Universal Robots PolyScope program: zaboj_fiala_program.urp

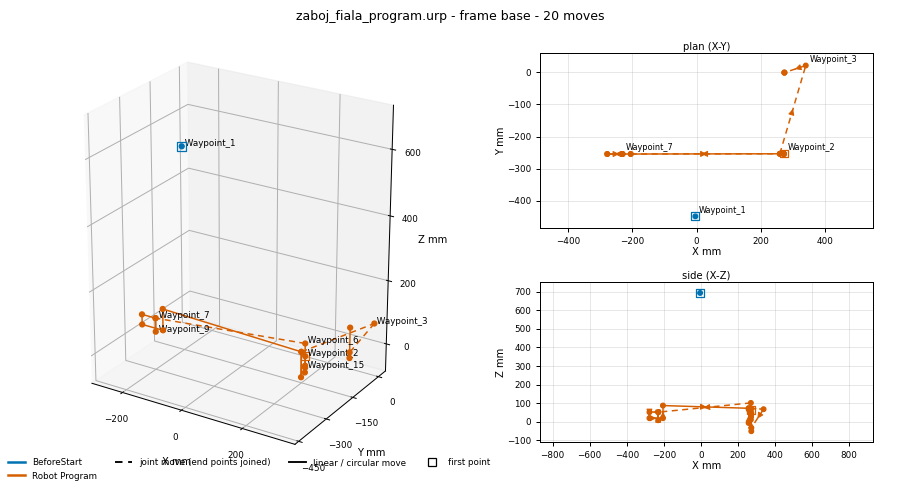
[picture p0: tool path of zaboj_fiala_program.urp in frame base, 20 of 20 moves have a stored position in this frame; points joined in program order, loops and branches not executed]
Program zaboj_fiala_program (installation=zaboj_fiala_instalace directory=/programs/usbdisk_0/new folder createdIn=5.21.2 lastSavedIn=5.21.2 robotSerialNumber=20185300578)
Calibrated DH parameters: a=[-0.000189, -0.243548, -0.212949, 0.000139, -0.000171, 0]; d=[0.151928, 2.340352, -3.79233, 1.582506, 0.085299, 0.092103]; alpha=[1.570802, 0.003282, -0.008312, 1.570809, -1.571939, 0]; deltaTheta=[0, 0.031526, 6.30827, -0.05661, 0, 0]
InitVariablesNode variables(variable(name=Pallet_1_cnt, expression=1), variable(name=Pallet_1_lct, expression=1), variable(name=Pallet_1_lno, expression=1), variable(name=Pallet_1_sep, expression=False), variable(name=Pallet_1_tct, expression=1), variable(name=qNearApproach, expression=[0,0,0,0,0,0]))
BeforeStart
  URCap Gripper Activate (Robotiq_Grippers, Robotiq Inc.) dataModel(ResetAndActivateKey=true)
  MoveJ speed 60 deg/s, acceleration 80 deg/s^2 (useActiveTCP=true optimoveEnabled=false optiMoveSpeed=0.3 optiMoveAcceleration=0.09) feature=Base
    Waypoint Waypoint_1: TCP in base x=-3.732 y=-447.764 z=694.669 mm, rx=0.0104 ry=2.2175 rz=-2.2154 rad; joints [0.253, -89.95, 0.625, -89.448, -0.524, -0.516] deg; TCP offset x=0.341 y=-0.738 z=225.168 mm, rx=0 ry=0 rz=-0.0028 rad
  Wait DigitalInput pin=digital_in[2]; digitalValue=1
Robot Program (runOnlyOnce=false)
  MoveJ speed 60 deg/s, acceleration 80 deg/s^2 (useActiveTCP=true optimoveEnabled=false optiMoveSpeed=0.3 optiMoveAcceleration=0.09) feature=Base
    Waypoint Waypoint_2: TCP in base x=270.562 y=-252.46 z=60.751 mm, rx=-2.2056 ry=2.2371 rz=0 rad; joints [-22.23, -101.243, -82.016, -86.674, 89.555, -21.444] deg
  Wait DigitalInput pin=digital_in[2]; digitalValue=1
  URCap Gripper (Robotiq_Grippers, Robotiq Inc.) dataModel(position=100.0, force=20.0, speed=100.0, positionInDouble=100.0, forceInDouble=20.0, speedInDouble=100.0, slaveIds=[9], blocking=true, robotCompliant=false)
  MoveL speed 50 mm/s, acceleration 1200 mm/s^2 (useActiveTCP=true optimoveEnabled=false optiMoveSpeed=0.01 optiMoveAcceleration=0.0001) feature=Base
    Waypoint Waypoint_15: TCP in base x=270.562 y=-252.46 z=25.108 mm, rx=-2.2056 ry=2.2371 rz=0 rad; joints [-22.21, -102.437, -90.223, -77.272, 89.565, -21.501] deg; TCP offset x=0.341 y=-0.738 z=225.168 mm, rx=0 ry=0 rz=-0.0028 rad
    var_1 := force()
    MoveL speed 250 mm/s, acceleration 1200 mm/s^2 (useActiveTCP=true optimoveEnabled=false optiMoveSpeed=0.3 optiMoveAcceleration=0.09) feature=Base
      Waypoint Waypoint_4: TCP in base x=271.723 y=-254.714 z=32.577 mm, rx=-2.2024 ry=2.234 rz=-0.0171 rad; joints [-22.478, -101.846, -89.192, -78.218, 89.558, -21.757] deg; TCP offset x=0.341 y=-0.738 z=225.168 mm, rx=0 ry=0 rz=-0.0028 rad
    If var_1>5
      MoveL speed 250 mm/s, acceleration 1200 mm/s^2 (useActiveTCP=true optimoveEnabled=false optiMoveSpeed=0.3 optiMoveAcceleration=0.09) feature=Base
        URCap Gripper (Robotiq_Grippers, Robotiq Inc.) dataModel(position=0.0, force=20.0, speed=100.0, positionInDouble=0.0, forceInDouble=20.0, speedInDouble=100.0, slaveIds=[9], blocking=true, robotCompliant=false)
        Waypoint Waypoint_5: TCP in base x=270.562 y=-253.262 z=10.468 mm, rx=-2.2056 ry=2.2371 rz=0 rad; joints [-22.326, -103.45, -93.013, -73.469, 89.574, -21.647] deg; TCP offset x=0.341 y=-0.738 z=225.168 mm, rx=0 ry=0 rz=-0.0028 rad
        URCap Gripper (Robotiq_Grippers, Robotiq Inc.) dataModel(position=100.0, force=20.0, speed=100.0, positionInDouble=100.0, forceInDouble=20.0, speedInDouble=100.0, slaveIds=[9], blocking=true, robotCompliant=false)
        SetPayload (workpieceName=Payload_brick payloadTransitionTime=0.05)
        Waypoint Waypoint_6: TCP in base x=270.562 y=-253.262 z=100.61 mm, rx=-2.2056 ry=2.2371 rz=0 rad; joints [-22.379, -101.712, -70.714, -97.506, 89.565, -21.504] deg
      MoveJ speed 60 deg/s, acceleration 80 deg/s^2 (useActiveTCP=true optimoveEnabled=false optiMoveSpeed=0.3 optiMoveAcceleration=0.09) feature=Base
        Waypoint Waypoint_7: TCP in base x=-230.059 y=-254.189 z=50.546 mm, rx=-2.2056 ry=2.2371 rz=0 rad; joints [-109.77, -94.859, -92.164, -82.912, 89.537, -109.018] deg
      MoveL speed 250 mm/s, acceleration 1200 mm/s^2 (useActiveTCP=true optimoveEnabled=false optiMoveSpeed=0.3 optiMoveAcceleration=0.09) feature=Base
        Waypoint Waypoint_9: TCP in base x=-230.059 y=-254.189 z=7.047 mm, rx=-2.2056 ry=2.2371 rz=0 rad; joints [-109.748, -97.199, -101.559, -71.177, 89.561, -109.091] deg
        URCap Gripper (Robotiq_Grippers, Robotiq Inc.) dataModel(position=0.0, force=100.0, speed=20.0, positionInDouble=0.0, forceInDouble=100.0, speedInDouble=20.0, slaveIds=[9], blocking=true, robotCompliant=false)
        SetPayload (workpieceName=Payload_Empty payloadTransitionTime=0.05)
        Waypoint Waypoint_7: TCP in base x=-230.059 y=-254.189 z=50.546 mm, rx=-2.2056 ry=2.2371 rz=0 rad; joints [-109.77, -94.859, -92.164, -82.912, 89.537, -109.018] deg
        URCap Gripper (Robotiq_Grippers, Robotiq Inc.) dataModel(position=100.0, force=100.0, speed=100.0, positionInDouble=100.0, forceInDouble=100.0, speedInDouble=100.0, slaveIds=[9], blocking=true, robotCompliant=false)
        MoveL speed 250 mm/s, acceleration 1200 mm/s^2 (useActiveTCP=true optimoveEnabled=false optiMoveSpeed=0.3 optiMoveAcceleration=0.09) feature=Base
          Waypoint Waypoint_11: motionParameters(blendRadius=0.01); TCP in base x=-277.401 y=-254.189 z=50.546 mm, rx=-2.2056 ry=2.2371 rz=0 rad; joints [-117.208, -103.279, -82.236, -84.42, 89.564, -116.439] deg
          Waypoint Waypoint_12: motionParameters(blendRadius=0.01); TCP in base x=-277.401 y=-254.189 z=18.071 mm, rx=-2.2056 ry=2.2371 rz=0 rad; joints [-117.19, -104.607, -89.405, -75.923, 89.576, -116.491] deg
          Waypoint Waypoint_13: motionParameters(blendRadius=0.01); TCP in base x=-204.474 y=-254.189 z=18.071 mm, rx=-2.2056 ry=2.2371 rz=0 rad; joints [-105.212, -92.223, -103.906, -73.805, 89.539, -104.534] deg
          Waypoint Waypoint_14: TCP in base x=-204.474 y=-254.189 z=86.413 mm, rx=-2.2056 ry=2.2371 rz=0 rad; joints [-105.25, -90.231, -87.365, -92.339, 89.523, -104.42] deg
    Else 
      MoveL speed 250 mm/s, acceleration 1200 mm/s^2 (useActiveTCP=true optimoveEnabled=false optiMoveSpeed=0.3 optiMoveAcceleration=0.09) feature=Base
        Waypoint Waypoint_8: TCP in base x=258.569 y=-253.444 z=71.606 mm, rx=-2.2024 ry=2.2403 rz=0 rad; joints [-23.165, -99.113, -81.653, -89.166, 89.548, -22.194] deg
        URCap Gripper (Robotiq_Grippers, Robotiq Inc.) dataModel(position=0.0, force=100.0, speed=20.0, positionInDouble=0.0, forceInDouble=100.0, speedInDouble=20.0, slaveIds=[9], blocking=true, robotCompliant=false)
        Waypoint Waypoint_10: TCP in base x=258.569 y=-253.444 z=-7.836 mm, rx=-2.2024 ry=2.2403 rz=0 rad; joints [-23.123, -102.847, -98.995, -68.09, 89.585, -22.323] deg; TCP offset x=0.341 y=-0.738 z=225.168 mm, rx=0 ry=0 rz=-0.0028 rad
        URCap Gripper (Robotiq_Grippers, Robotiq Inc.) dataModel(position=100.0, force=100.0, speed=20.0, positionInDouble=100.0, forceInDouble=100.0, speedInDouble=20.0, slaveIds=[9], blocking=true, robotCompliant=false)
        SetPayload (workpieceName=Payload_brick payloadTransitionTime=0.05)
        Waypoint Waypoint_8: TCP in base x=258.569 y=-253.444 z=71.606 mm, rx=-2.2024 ry=2.2403 rz=0 rad; joints [-23.165, -99.113, -81.653, -89.166, 89.548, -22.194] deg; TCP offset x=0.341 y=-0.738 z=225.168 mm, rx=0 ry=0 rz=-0.0028 rad
        MoveJ speed 60 deg/s, acceleration 80 deg/s^2 (useActiveTCP=true optimoveEnabled=false optiMoveSpeed=0.3 optiMoveAcceleration=0.09) feature=Base
          Waypoint Waypoint_3: TCP in base x=339.173 y=20.646 z=66.699 mm, rx=-0.0469 ry=3.1402 rz=-0.0152 rad; joints [26.842, -93.739, -88.951, -87.435, 89.002, 115.109] deg; TCP offset x=0.341 y=-0.738 z=225.168 mm, rx=0 ry=0 rz=-0.0028 rad
        URCap Palletizing (polyscope-pallet-impl, Universal Robots) dataModel(palletFeature=Base, isPalletizing=true, Variable(key=qNearApproach, variable(name=qNearApproach, initializeExpression=[0,0,0,0,0,0])), Variable(key=name, variable(name=Pallet_1)), Variable(key=globalCountingVariable, variable(name=Pallet_1_cnt, initializeExpression=1)), Variable(key=layerNumberVariable, variable(name=Pallet_1_lno, initializeExpression=1)), Variable(key=layerCountingVariable, variable(name=Pallet_1_lct, initializeExpression=1)), Variable(key=handleSeparatorVariable, variable(name=Pallet_1_sep, initializeExpression=False)), Variable(key=totalCountVariable, variable(name=Pallet_1_tct, initializeExpression=1)), Length(key=objectHeight value=0.029 unit=M), Variable(key=referencePoint, variable(featureName=referencePoint)), Variable(key=separatorPoint, variable(featureName=separatorPoint))); state(isChildrenLocked=true)
          URCap Patterns (polyscope-pallet-impl, Universal Robots) state(isChildrenLocked=true)
            URCap Pattern (polyscope-pallet-impl, Universal Robots) dataModel(UUID=fb6f7ec9-a042-4793-b577-05f4db72c464, patternType=GRID, columns=2, rows=3, Variable(key=nameVariable, variable(name=Grid_Pattern_1))); state(isChildrenLocked=true)
              URCap Item (polyscope-pallet-impl, Universal Robots) dataModel(UUID=009ec79f-ed00-48c4-8bc6-377c492b1326, patternType=GRID, index=0, calibrationDeltaTheta=[-9.679944364821003E-8, 0.03152637960071048, 6.308270136326222, -0.05660981424064361, 2.1302738175549285E-7, -3.4337321612454286E-7], calibrationA=[-1.89170984734602E-4, -0.24354794633452972, -0.2129485167088614, 1.3892904611349137E-4, -1.7067015336856014E-4, 0.0], calibrationD=[0.15192760230984942, 2.3403518756598336, -3.792330157129607, 1.5825055280731988, 0.08529876240250026, 0.09210299655971649], calibrationAlpha=[1.5708023866418512, 0.0032819461853986743, -0.008311935193061136, 1.570808769909054, -1.5719389687286305, 0.0], calibrationJointChecksum=[-1323472732, -1322302140, 655890344, -1781272900, -1781497016, -1329631202], calibrationStatus=2, calibrationValidChecksum=true, baseToFeature=[0.0, 0.0, 0.0, 0.0, 0.0, 0.0], TCPOffset=[3.5168318263162357E-4, -7.609358326787711E-4, 0.2251763575477216, -1.1367748142535932E-5, 2.2048030494940052E-5, -0.0027178388032577955], Variable(key=variable, variable(name=CornerItem_1)), JointPositions(key=jointpositions, JointPosition(key=[1], Angle(key=pos value=0.50025 unit=RAD)), JointPosition(key=[2], Angle(key=pos value=-1.512423 unit=RAD)), JointPosition(key=[3], Angle(key=pos value=-2.280893 unit=RAD)), JointPosition(key=[4], Angle(key=pos value=-0.917942 unit=RAD)), JointPosition(key=[5], Angle(key=pos value=1.563579 unit=RAD)), JointPosition(key=[6], Angle(key=pos value=2.060299 unit=RAD))))
              URCap Item (polyscope-pallet-impl, Universal Robots) dataModel(UUID=98a13d22-f757-4477-b5d1-566cbffb46b7, patternType=GRID, index=1, calibrationDeltaTheta=[-9.679944364821003E-8, 0.03152637960071048, 6.308270136326222, -0.05660981424064361, 2.1302738175549285E-7, -3.4337321612454286E-7], calibrationA=[-1.89170984734602E-4, -0.24354794633452972, -0.2129485167088614, 1.3892904611349137E-4, -1.7067015336856014E-4, 0.0], calibrationD=[0.15192760230984942, 2.3403518756598336, -3.792330157129607, 1.5825055280731988, 0.08529876240250026, 0.09210299655971649], calibrationAlpha=[1.5708023866418512, 0.0032819461853986743, -0.008311935193061136, 1.570808769909054, -1.5719389687286305, 0.0], calibrationJointChecksum=[-1323472732, -1322302140, 655890344, -1781272900, -1781497016, -1329631202], calibrationStatus=2, calibrationValidChecksum=true, baseToFeature=[0.0, 0.0, 0.0, 0.0, 0.0, 0.0], TCPOffset=[3.41180420217968E-4, -7.536512495878241E-4, 0.22516676469490038, -2.730457853376625E-5, -2.5939791816466612E-5, -0.002754566285013443], Variable(key=variable, variable(name=CornerItem_2)), JointPositions(key=jointpositions, JointPosition(key=[1], Angle(key=pos value=0.342042 unit=RAD)), JointPosition(key=[2], Angle(key=pos value=-1.996811 unit=RAD)), JointPosition(key=[3], Angle(key=pos value=-1.683961 unit=RAD)), JointPosition(key=[4], Angle(key=pos value=-1.03053 unit=RAD)), JointPosition(key=[5], Angle(key=pos value=1.564631 unit=RAD)), JointPosition(key=[6], Angle(key=pos value=1.903189 unit=RAD))))
              URCap Item (polyscope-pallet-impl, Universal Robots) dataModel(UUID=f0fdfe4c-2f28-4653-b719-23e1e8829ea8, patternType=GRID, index=2, calibrationDeltaTheta=[-9.679944364821003E-8, 0.03152637960071048, 6.308270136326222, -0.05660981424064361, 2.1302738175549285E-7, -3.4337321612454286E-7], calibrationA=[-1.89170984734602E-4, -0.24354794633452972, -0.2129485167088614, 1.3892904611349137E-4, -1.7067015336856014E-4, 0.0], calibrationD=[0.15192760230984942, 2.3403518756598336, -3.792330157129607, 1.5825055280731988, 0.08529876240250026, 0.09210299655971649], calibrationAlpha=[1.5708023866418512, 0.0032819461853986743, -0.008311935193061136, 1.570808769909054, -1.5719389687286305, 0.0], calibrationJointChecksum=[-1323472732, -1322302140, 655890344, -1781272900, -1781497016, -1329631202], calibrationStatus=2, calibrationValidChecksum=true, baseToFeature=[0.0, 0.0, 0.0, 0.0, 0.0, 0.0], TCPOffset=[3.40518158797376E-4, -7.536866787021881E-4, 0.22516907041249068, -4.076573333353527E-6, -4.229667960397262E-6, -0.002774856931555885], Variable(key=variable, variable(name=CornerItem_3)), JointPositions(key=jointpositions, JointPosition(key=[1], Angle(key=pos value=0.499268 unit=RAD)), JointPosition(key=[2], Angle(key=pos value=-2.012468 unit=RAD)), JointPosition(key=[3], Angle(key=pos value=-1.65953 unit=RAD)), JointPosition(key=[4], Angle(key=pos value=-1.039312 unit=RAD)), JointPosition(key=[5], Angle(key=pos value=1.564656 unit=RAD)), JointPosition(key=[6], Angle(key=pos value=2.060499 unit=RAD))))
              URCap Item (polyscope-pallet-impl, Universal Robots) dataModel(UUID=1b0446d0-c541-46d0-9146-9f7b7f3340ef, patternType=GRID, index=3, calibrationDeltaTheta=[-9.679944364821003E-8, 0.03152637960071048, 6.308270136326222, -0.05660981424064361, 2.1302738175549285E-7, -3.4337321612454286E-7], calibrationA=[-1.89170984734602E-4, -0.24354794633452972, -0.2129485167088614, 1.3892904611349137E-4, -1.7067015336856014E-4, 0.0], calibrationD=[0.15192760230984942, 2.3403518756598336, -3.792330157129607, 1.5825055280731988, 0.08529876240250026, 0.09210299655971649], calibrationAlpha=[1.5708023866418512, 0.0032819461853986743, -0.008311935193061136, 1.570808769909054, -1.5719389687286305, 0.0], calibrationJointChecksum=[-1323472732, -1322302140, 655890344, -1781272900, -1781497016, -1329631202], calibrationStatus=2, calibrationValidChecksum=true, baseToFeature=[0.0, 0.0, 0.0, 0.0, 0.0, 0.0], TCPOffset=[3.4398629409498893E-4, -7.549386560833996E-4, 0.22517806179782512, -1.7407097723726922E-5, 1.2818392060821723E-5, -0.0027473222426862764], Variable(key=variable, variable(name=CornerItem_4)), JointPositions(key=jointpositions, JointPosition(key=[1], Angle(key=pos value=0.716646 unit=RAD)), JointPosition(key=[2], Angle(key=pos value=-1.550889 unit=RAD)), JointPosition(key=[3], Angle(key=pos value=-2.259742 unit=RAD)), JointPosition(key=[4], Angle(key=pos value=-0.900677 unit=RAD)), JointPosition(key=[5], Angle(key=pos value=1.563789 unit=RAD)), JointPosition(key=[6], Angle(key=pos value=2.276623 unit=RAD))))
          URCap Layers (polyscope-pallet-impl, Universal Robots) dataModel(separators=[false], selectedPatterns=[fb6f7ec9-a042-4793-b577-05f4db72c464])
          URCap At Each Item (polyscope-pallet-impl, Universal Robots) dataModel(selectedPattern=fb6f7ec9-a042-4793-b577-05f4db72c464, selectedPosition=009ec79f-ed00-48c4-8bc6-377c492b1326, currentWizardState=MANUAL, Pose(key=refBaseToFeature, Position(key=posePosition, Length(key=X value=0 unit=M), Length(key=Y value=0 unit=M), Length(key=Z value=0 unit=M)), Rotation(key=poseRotation, Angle(key=RX value=0 unit=RAD), Angle(key=RY value=0 unit=RAD), Angle(key=RZ value=0 unit=RAD))), Pose(key=refPose, Position(key=posePosition, Length(key=X value=0.272815 unit=M), Length(key=Y value=-0.001325 unit=M), Length(key=Z value=-0.052174 unit=M)), Rotation(key=poseRotation, Angle(key=RX value=0.008705 unit=RAD), Angle(key=RY value=-3.14155 unit=RAD), Angle(key=RZ value=0.000049 unit=RAD))))
            URCap Generated Movements (polyscope-pallet-impl, Universal Robots) state(isChildrenLocked=true)
              MoveJ speed 60 deg/s, acceleration 80 deg/s^2 (useActiveTCP=true optimoveEnabled=false optiMoveSpeed=0.3 optiMoveAcceleration=0.09) feature=referencePoint
                Waypoint Approach: TCP in base x=272.815 y=-1.325 z=-33.906 mm, rx=0.0087 ry=-3.1415 rz=0 rad; joints [28.649, -83.512, -127.496, -58.93, 89.548, 118.083] deg; feature pose in base x=272.815 y=-1.325 z=-52.174 mm, rx=0.0087 ry=-3.1415 rz=0 rad
              MoveL speed 250 mm/s, acceleration 1200 mm/s^2 (useActiveTCP=true optimoveEnabled=false optiMoveSpeed=0.3 optiMoveAcceleration=0.09) feature(featureName=referencePoint)
                Waypoint ToolActionPoint: TCP in base x=272.816 y=-1.325 z=-52.174 mm, rx=0.0087 ry=-3.1416 rz=0 rad; joints [28.662, -86.655, -130.686, -52.594, 89.586, 118.046] deg; TCP offset x=0.352 y=-0.761 z=225.176 mm, rx=0 ry=0 rz=-0.0027 rad
              Folder Tool action
                URCap Gripper (Robotiq_Grippers, Robotiq Inc.) dataModel(position=0.0, force=100.0, speed=20.0, positionInDouble=0.0, forceInDouble=100.0, speedInDouble=20.0, slaveIds=[9], blocking=true, robotCompliant=false)
                SetPayload (workpieceName=Payload_Empty payloadTransitionTime=0.05)
              MoveL speed 250 mm/s, acceleration 1200 mm/s^2 (useActiveTCP=true optimoveEnabled=false optiMoveSpeed=0.3 optiMoveAcceleration=0.09) feature(featureName=referencePoint)
                Waypoint Exit_1: TCP in base x=272.815 y=-1.325 z=45.468 mm, rx=0.0087 ry=-3.1416 rz=0 rad; joints [28.605, -76.502, -110.272, -83.164, 89.472, 118.236] deg; TCP offset x=0.341 y=-0.738 z=225.168 mm, rx=0 ry=0 rz=-0.0028 rad
Thread Thread_1 (runOnlyOnce=false)
  Set DigitalOutput pin=digital_out[2]; digitalValue=1
  Wait DigitalInput pin=digital_in[2]; digitalValue=1
  Set DigitalOutput pin=digital_out[2]; digitalValue=0
  Wait DigitalInput pin=digital_in[2]; digitalValue=0
  Wait Sleep waitTime=1
